{attribute 'GeneratedUsingTerminal: EK1122-0000-0018'}
{attribute addProperty BoxType "EK1122-0000-0018"}
{attribute addProperty Id "Beckhoff_EP1xxxsub_EK1100EK1100_1FC0878B2A_0001_EP1008_0001_0016EP1008_78E8D3DD12A_0002_EP1008_0001_0017EP1008_78E8D3DD12A_0003_EP1008_0001_0018EP1008_78E8D3DD12A_0004_EP1008_0002_0016EP1008_78E8D3DD12A_0005_EP1008_0002_0017EP1008_78E8D3DD12A_0006_EP1008_0002_0018EP1008_78E8D3DD12A_0007_EP1008_0022_0016EP1008_78E8D3DD12A_0008_EP1008_0022_0017EP1008_78E8D3DD12A_0009_EP1018_0001_0016EP1018_78E8D3DD12A_0010_EP1018_0001_0017EP1018_78E8D3DD12A_0011_EP1018_0001_0018EP1018_78E8D3DD12A_0012_EP1018_0401_0016EP1018_78E8D3DD12A_0013_EP1018_0002_0016EP1018_78E8D3DD12A_0014_EP1018_0002_0017EP1018_78E8D3DD12A_0015_EP1018_0002_0018EP1018_78E8D3DD12A_0016_EP1098_0001_0016EP1098_78E8D3DD12A_0017_EP1098_0001_0017EP1098_78E8D3DD12A_0018_EP1111_0000_0016EP1111_837A6B0314A_0019_EP1111_0000_0017EP1111_837A6B0314A_0020_EP1111_0000_0018EP1111_837A6B0314A_0021_EP1111_0000_0019EP1111_837A6B0314A_0022_EP1111_0000_0020EP1111_837A6B0314A_0023_EP1111_0000_0021EP1111_837A6B0314A_0024_EP1122_0001_0016A_0024_EP1122_0001_0016_DB5F1CD01450"}
{attribute addProperty CRC "861395881"}
{attribute addProperty Size "1740"}
{attribute addProperty Name "Beckhoff EP1xxxEK1122"}
TYPE Beckhoff_EP1xxxEK1122_3357DBA9 EXTENDS EK1122_1FC0878B :
STRUCT
	{attribute addProperty Name "Beckhoff EP1xxxsub EK1100"}
	{attribute addProperty PreviousPort "Beckhoff EP1xxxEK1122 : D"}
	Beckhoff_EP1xxxsub_EK1100 : EK1100_1FC0878B;
	{attribute addProperty Name "A_0001(EP1008-0001-0016)"}
	{attribute addProperty PreviousPort "Beckhoff EP1xxxsub EK1100 : C"}
	A_0001_EP1008_0001_0016 : EP1008_78E8D3DD;
	{attribute addProperty Name "A_0002(EP1008-0001-0017)"}
	{attribute addProperty PreviousPort "A_0001(EP1008-0001-0016) : B"}
	A_0002_EP1008_0001_0017 : EP1008_78E8D3DD;
	{attribute addProperty Name "A_0003(EP1008-0001-0018)"}
	{attribute addProperty PreviousPort "A_0002(EP1008-0001-0017) : B"}
	A_0003_EP1008_0001_0018 : EP1008_78E8D3DD;
	{attribute addProperty Name "A_0004(EP1008-0002-0016)"}
	{attribute addProperty PreviousPort "A_0003(EP1008-0001-0018) : B"}
	A_0004_EP1008_0002_0016 : EP1008_78E8D3DD;
	{attribute addProperty Name "A_0005(EP1008-0002-0017)"}
	{attribute addProperty PreviousPort "A_0004(EP1008-0002-0016) : B"}
	A_0005_EP1008_0002_0017 : EP1008_78E8D3DD;
	{attribute addProperty Name "A_0006(EP1008-0002-0018)"}
	{attribute addProperty PreviousPort "A_0005(EP1008-0002-0017) : B"}
	A_0006_EP1008_0002_0018 : EP1008_78E8D3DD;
	{attribute addProperty Name "A_0007(EP1008-0022-0016)"}
	{attribute addProperty PreviousPort "A_0006(EP1008-0002-0018) : B"}
	A_0007_EP1008_0022_0016 : EP1008_78E8D3DD;
	{attribute addProperty Name "A_0008(EP1008-0022-0017)"}
	{attribute addProperty PreviousPort "A_0007(EP1008-0022-0016) : B"}
	A_0008_EP1008_0022_0017 : EP1008_78E8D3DD;
	{attribute addProperty Name "A_0009(EP1018-0001-0016)"}
	{attribute addProperty PreviousPort "A_0008(EP1008-0022-0017) : B"}
	A_0009_EP1018_0001_0016 : EP1018_78E8D3DD;
	{attribute addProperty Name "A_0010(EP1018-0001-0017)"}
	{attribute addProperty PreviousPort "A_0009(EP1018-0001-0016) : B"}
	A_0010_EP1018_0001_0017 : EP1018_78E8D3DD;
	{attribute addProperty Name "A_0011(EP1018-0001-0018)"}
	{attribute addProperty PreviousPort "A_0010(EP1018-0001-0017) : B"}
	A_0011_EP1018_0001_0018 : EP1018_78E8D3DD;
	{attribute addProperty Name "A_0012(EP1018-0401-0016)"}
	{attribute addProperty PreviousPort "A_0011(EP1018-0001-0018) : B"}
	A_0012_EP1018_0401_0016 : EP1018_78E8D3DD;
	{attribute addProperty Name "A_0013(EP1018-0002-0016)"}
	{attribute addProperty PreviousPort "A_0012(EP1018-0401-0016) : B"}
	A_0013_EP1018_0002_0016 : EP1018_78E8D3DD;
	{attribute addProperty Name "A_0014(EP1018-0002-0017)"}
	{attribute addProperty PreviousPort "A_0013(EP1018-0002-0016) : B"}
	A_0014_EP1018_0002_0017 : EP1018_78E8D3DD;
	{attribute addProperty Name "A_0015(EP1018-0002-0018)"}
	{attribute addProperty PreviousPort "A_0014(EP1018-0002-0017) : B"}
	A_0015_EP1018_0002_0018 : EP1018_78E8D3DD;
	{attribute addProperty Name "A_0016(EP1098-0001-0016)"}
	{attribute addProperty PreviousPort "A_0015(EP1018-0002-0018) : B"}
	A_0016_EP1098_0001_0016 : EP1098_78E8D3DD;
	{attribute addProperty Name "A_0017(EP1098-0001-0017)"}
	{attribute addProperty PreviousPort "A_0016(EP1098-0001-0016) : B"}
	A_0017_EP1098_0001_0017 : EP1098_78E8D3DD;
	{attribute addProperty Name "A_0018(EP1111-0000-0016)"}
	{attribute addProperty PreviousPort "A_0017(EP1098-0001-0017) : B"}
	A_0018_EP1111_0000_0016 : EP1111_837A6B03;
	{attribute addProperty Name "A_0019(EP1111-0000-0017)"}
	{attribute addProperty PreviousPort "A_0018(EP1111-0000-0016) : B"}
	A_0019_EP1111_0000_0017 : EP1111_837A6B03;
	{attribute addProperty Name "A_0020(EP1111-0000-0018)"}
	{attribute addProperty PreviousPort "A_0019(EP1111-0000-0017) : B"}
	A_0020_EP1111_0000_0018 : EP1111_837A6B03;
	{attribute addProperty Name "A_0021(EP1111-0000-0019)"}
	{attribute addProperty PreviousPort "A_0020(EP1111-0000-0018) : B"}
	A_0021_EP1111_0000_0019 : EP1111_837A6B03;
	{attribute addProperty Name "A_0022(EP1111-0000-0020)"}
	{attribute addProperty PreviousPort "A_0021(EP1111-0000-0019) : B"}
	A_0022_EP1111_0000_0020 : EP1111_837A6B03;
	{attribute addProperty Name "A_0023(EP1111-0000-0021)"}
	{attribute addProperty PreviousPort "A_0022(EP1111-0000-0020) : B"}
	A_0023_EP1111_0000_0021 : EP1111_837A6B03;
	{attribute addProperty Name "A_0024(EP1122-0001-0016)"}
	{attribute addProperty PreviousPort "A_0023(EP1111-0000-0021) : B"}
	A_0024_EP1122_0001_0016 : A_0024_EP1122_0001_0016_DB5F1CD0;
END_STRUCT
END_TYPE

(* stored: Version 1.2.0.0, ProductVersion 3.1.4024.11
   DUT Beckhoff_EP1xxxEK1122_3357DBA9: Id {49b58939-c16c-43fc-bece-d0b0ebcdfc7f} *)
